# EPICS autosave request: ADApp/Db/NDArrayBase_settings.req
$(P)$(R)DataType
$(P)$(R)ColorMode
$(P)$(R)ArrayCallbacks
$(P)$(R)NDAttributesFile
$(P)$(R)NDAttributesMacros
$(P)$(R)PoolUsedMem.SCAN
